// CALCULATE NEXT STEAM TEMPURATURE

FUNCTION RunSteam

VAR
	
	// User input target
	targ : REAL := userin.steam_temp;
	enabled : bool := userin.enable_steam;
	
	// Import steam parameters for clarity
	now  : REAL := steam.now;
	maxi : REAL := steam.maxi;
	mini : REAL := steam.mini;
	step : REAL := steam.step * userin.time_step;
	
	// Calculation variables
	new  : REAL;
	diff : REAL;
	
END_VAR

// Import target temp from GUI
steam.target := targ;

// Validation
IF step <= 0 THEN
	RETURN;
ELSIF targ > maxi THEN
	targ := maxi;
ELSIF targ < mini THEN
	targ := mini;
END_IF

// Manual override
IF NOT enabled THEN
	targ := 20;
END_IF


// Calculate what change is needed to meet the target
diff := targ - now;


// LESS than target and MORE than a step away
IF diff >= step THEN
	// New temp is this plus step
	new := now + step;	

// GREATER then target and MORE than a step away
ELSIF diff <= -step THEN
	// New temp is this minus step
	new := now - step;

// Is correct or within one step
ELSE
	new := targ;
END_IF

// Save new value
temp.wall := new;
steam.now := new;

END_FUNCTION

(* stored: Version 1.1.0.1, ProductVersion 3.1.4024.12
   POU RunSteam: Id {475fa9dc-9a0d-4478-a41e-ad86e1ec38db}, SpecialFunc None *)
